PROGRAM P_EnOcean
VAR
	fbKL6581			: FB_KL6581;
	stKL6581_in  AT %I* : KL6581_INPUT;
	stKL6581_out AT %Q*	: KL6581_OUTPUT;
	stKL6581			: STR_KL6581;
	bInitCom			: BOOL := TRUE;
	
	arrEnOcean_Search	: ARRAY [1..8] OF FB_EnOcean_Search;
	nSearchIdx			: BYTE;
	bSerach				: BOOL;
	arrDevices			: ARRAY [1..8] OF INT;
	arrID				: ARRAY [1..8, 0..255] OF DWORD;
	
		//Trykknapper Atrium
	fbGang_3_109_Kantine_Tryk_PladeA     	: FB_Rec_RPS_Switch;
	fbAtriumNiveau_Tryk_PladeB				: FB_Rec_RPS_Switch;
	fbAtriumNiveau_Tryk_Sevice				: FB_Rec_RPS_Switch;
	//Trykknapper på gange
	fbGang_7_301_Tryk			: FB_Rec_RPS_Switch;
	
	//Trykknapper i rum
	fbRum_2_341_Tryk_Indgang		: FB_Rec_RPS_Switch;
	fbRum_2_341_Tryk_Ekstra			: FB_Rec_RPS_Switch;
	fbRum_2_345_Tryk                : FB_Rec_RPS_Switch;
	fbRum_2_345_Tryk_Ekstra			: FB_Rec_RPS_Switch;
	fbRum_2_349_Tryk				: FB_Rec_RPS_Switch;
	
END_VAR

VAR CONSTANT
	byNode_1: BYTE := 1;
	byNode_2: BYTE := 2;
	byNode_3: BYTE := 3;
	byNode_4: BYTE := 4;
	byNode_5: BYTE := 5;
	byNode_6: BYTE := 6;
	byNode_7: BYTE := 7;
	byNode_8: BYTE := 8;
END_VAR


(* Kommunikation mit der KL6581. *)
(* Communication with the KL6581. *)
fbKL6581(
	bInit			:= bInitCom,
	nIdx			:= 2,
	stKL6581_in		:= stKL6581_In,
	stKL6581_out	:= stKL6581_Out,
	bReady			=> ,
	bBusy			=> ,
	bError			=> ,
	iErrorID		=> ,
	str_KL6581		=> stKL6581);

(* Warten bis der Kommunikationsbaustein initialisiert wurde.*)
(* Wait until the communication function block has been initialized. *)
IF (NOT fbKL6581.bReady) THEN
	RETURN;
END_IF

FOR nSearchIdx:= 1 TO 8 DO
	arrEnOcean_Search[nSearchIdx](
		bStart:= TRUE, 
		str_KL6581:= stKL6581 , 
		byNode:= nSearchIdx, 
		bReceive=> , 
		iDevices=>arrDevices[nSearchIdx] , 
		ar_ID=> );
		
		MEMCPY(ADR(arrID[nSearchIdx,0]), ADR(arrEnOcean_Search[nSearchIdx].ar_ID), SIZEOF(arrEnOcean_Search[nSearchIdx].ar_ID)); 
END_FOR
//AtriumNiveau
A_AtriumNiveau();

A_Gang_7_301();

A_Rum_2_341();
A_Rum_2_345();
A_Rum_2_345_1();

ACTION A_AtriumNiveau:
fbAtriumNiveau_Tryk_PladeB(
	str_KL6581:=stKL6581 , 
	byNode:=0 , 
	dw_ID:= 16#0029B92D, 
	str_EnOceanSwitch=> GVL_EnOcean.strEnOceanSwitch_AtriumNiveau_PladeB,
	by_Node=> , 
	bReceive=> );


(*
fbAtriumNiveau_Tryk_PladeB(
	str_KL6581:=stKL6581 , 
	byNode:=0, 
	dw_ID:= 16#00FEE4FE87, 
	str_EnOceanSwitch=> GVL_EnOcean.strEnOceanSwitch_AtriumNiveau_Service, 
	by_Node=> , 
	bReceive=> );
	*)
END_ACTION

ACTION A_Gang_7_301:

fbGang_7_301_Tryk(
	str_KL6581:=stKL6581 , 
	byNode:= byNode_2, 
	dw_ID:= 16#21C437, 
	str_EnOceanSwitch=> GVL_EnOcean.strEnOceanSwitch_Gang_7_301, 
	by_Node=> , 
	bReceive=> );
END_ACTION

ACTION A_Rum_2_341:
fbRum_2_341_Tryk_Indgang(
	str_KL6581:=stKL6581 , 
	byNode:=byNode_2 , 
	dw_ID:= 16#2F2DAF, 
	str_EnOceanSwitch=> GVL_EnOcean.strEnOceanSwitch_Rum_2_341_Indgang, 
	by_Node=> , 
	bReceive=> );
	
	fbRum_2_341_Tryk_Ekstra(
	str_KL6581:=stKL6581 , 
	byNode:= byNode_2 , 
	dw_ID:= 16#29B92A, 
	str_EnOceanSwitch=> GVL_EnOcean.strEnOceanSwitch_Rum_2_341_Ekstra, 
	by_Node=> , 
	bReceive=> );
END_ACTION

ACTION A_Rum_2_345:

	
	fbRum_2_345_Tryk_Ekstra(
	str_KL6581:=stKL6581 , 
	byNode:= byNode_2 , 
	dw_ID:= 16#29B783, 
	str_EnOceanSwitch=> GVL_EnOcean.strEnOceanSwitch_Rum_2_345_Ekstra, 
	by_Node=> , 
	bReceive=> );
END_ACTION

ACTION A_Rum_2_345_1:

	
	fbRum_2_345_Tryk(
	str_KL6581:=stKL6581 , 
	byNode:= byNode_2 , 
	dw_ID:= 16#0029B97D, 
	str_EnOceanSwitch=> GVL_EnOcean.strEnOceanSwitch_Rum_2_345, 
	by_Node=> , 
	bReceive=> );
END_ACTION

END_PROGRAM

(* stored: Version 1.1.0.1
   POU P_EnOcean: Id {d2583012-7b8d-42b3-930e-7213eee0e992}, SpecialFunc None
   Action A_AtriumNiveau: Id {5b863a8e-6cff-4511-86bf-f0a83cf94e37}
   Action A_Gang_7_301: Id {8247182c-a772-4b27-815a-da064112dabc}
   Action A_Rum_2_341: Id {aeb6deef-b26d-4eb5-9023-a9a71a25ad64}
   Action A_Rum_2_345: Id {99aefd77-4d33-48e1-aeac-2b850a10feaa}
   Action A_Rum_2_345_1: Id {a81c6b92-747e-403b-95a8-34336932ba48} *)
